{attribute 'linkalways'} 
{attribute 'no_explicit_call' := 'This FB is a CLASS and must be accessed using methods or properties'}
{attribute 'enable_dynamic_creation'}
FUNCTION_BLOCK Node_F_VN_InsertIntoContainer_TcVnPoint3_REAL EXTENDS VisionNode
VAR
    aElement : _TcVnPoint3_REAL;
    ipContainer : _ITcVnContainer;
    nIndex : _ULINT(0);
    hrPrev : _HRESULT(S_OK);
    hresult : _HRESULT(S_OK);
END_VAR

METHOD PUBLIC  Clone : I_Node
VAR
	pNode : POINTER TO Node_F_VN_InsertIntoContainer_TcVnPoint3_REAL;
END_VAR
pNode := __NEW(Node_F_VN_InsertIntoContainer_TcVnPoint3_REAL);
Clone := pNode^;
END_METHOD

METHOD FB_init : BOOL
VAR_INPUT
	bInitRetains : BOOL; // if TRUE, the retain variables are initialized (warm start / cold start)
	bInCopyCode : BOOL;  // if TRUE, the instance afterwards gets moved into the copy code (online change)
END_VAR
AddInput('aElement', aElement);
AddInput('ipContainer', ipContainer);
AddInput('nIndex', nIndex);
AddInput('hrPrev', hrPrev);
AddOutput('ipContainer', ipContainer);
AddOutput('hresult',hresult);
END_METHOD

METHOD PROTECTED OnExecute : HRESULT
hresult.Value := F_VN_InsertIntoContainer_TcVnPoint3_REAL(
    aElement := aElement.Value,
    ipContainer := ipContainer.Value,
    nIndex := nIndex.Value,
    hrPrev:= hrPrev.Value);
END_METHOD

METHOD PUBLIC PreExecutionCheck
VAR_INPUT
	Check : I_PreExecutionChecks;
END_VAR
Check.IsTrue(ipContainer.IsValid, 'ipContainer must be a valid container');
END_METHOD

END_FUNCTION_BLOCK

(* stored: Version 1.1.0.1, ProductVersion 3.1.4024.13
   POU Node_F_VN_InsertIntoContainer_TcVnPoint3_REAL: Id {8f21e689-b97e-4f6a-931b-4e662d23a6f9}, SpecialFunc None
   Folder Constructor: Id {31b65fec-e061-427f-8e28-4837030e95d8}
   Method Clone: Id {cd2bf488-9141-4f61-9889-8f6832ee03ad}
   Method FB_init: Id {ad283df2-01b0-471d-90b4-9b30ca2c6cc6}
   Method OnExecute: Id {db321cf7-1eba-4023-ba64-38ec2b6e854b}
   Method PreExecutionCheck: Id {a7968650-d208-49d2-a49b-b05d108674c5} *)
